Universal Robots PolyScope program: Exercise2_easyprogramming.urp

Program Exercise2_easyprogramming (installation=default directory=/home/ur/ursim-current/programs createdIn=5.7.0.90932 lastSavedIn=5.7.0.90932 robotSerialNumber=20195599999)
Calibrated DH parameters: a=[0, -0.425, -0.3922, 0, 0, 0]; d=[0.1625, 0, 0, 0.1333, 0.0997, 0.0996]; alpha=[1.570796, 0, 0, 1.570796, -1.570796, 0]; deltaTheta=[0, 0, 0, 0, 0, 0]
Robot Program (runOnlyOnce=true)
  Popup Message (haltProgram=false message=Iniciando Programa inputType=Text)
  i := 0
  j := 0
  x := 0
  y := 0
  n_col := 3
  n_filas := 3
  dist := 0.1
  Set NoAction (payload=1.5 tcpAsCog=true) tcp=TCP
  MoveJ speed 60 deg/s, acceleration 80 deg/s^2 (useActiveTCP=true) feature=Base
    Waypoint Waypoint_1 (Variable): variable=safe_pose
    'Movimiento inicial'
  Loop While (checkContinuously=false) expression=i<n_filas
    Loop While (checkContinuously=false) expression=j<n_col
      pose_sig := p[0.5+x,-0.15+y,0.05,0,3.1416,0]
      pose_desb := p[0.5+x,-0.15+y,0,0,3.1416,0]
      'Movimiento de llegada y desbarbado'
      MoveJ speed 60 deg/s, acceleration 80 deg/s^2 (useActiveTCP=true) feature=Base
        Waypoint Waypoint_1 (Variable): variable=pose_sig
      MoveL speed 250 mm/s, acceleration 1200 mm/s^2 (useActiveTCP=true) feature=Base
        Waypoint Waypoint_1 (Variable): variable=pose_desb
      Wait Sleep waitTime=2.5
      MoveL speed 250 mm/s, acceleration 1200 mm/s^2 (useActiveTCP=true) feature=Base
        Waypoint Waypoint_1 (Variable): variable=pose_sig
      'Siguiente columna'
      y := y+dist
      j := j+1
    'Siguiente fila'
    i := i+1
    j := 0
    x := x+dist
    y := 0
  MoveJ speed 60 deg/s, acceleration 80 deg/s^2 (useActiveTCP=true) feature=Base
    Waypoint Waypoint_2 (Variable): variable=safe_pose
    'Vuelta a la posición de seguridad'
